// TIA Portal V17 export
// export: Created 2024-08-07T21:44:10.5201385Z, ExportSetting WithDefaults, DisplayName Totally Integrated Automation Portal, DisplayVersion V17 Update 7, DisplayName TIA Portal Openness, DisplayVersion V17 Update 7, DisplayName TIA Portal Version Control Interface, DisplayVersion V17, DisplayName SINAMICS Startdrive Advanced, DisplayVersion V17 SP2, DisplayName SINAMICS Startdrive G110M, G120, G120C, G120D, G120P, G115D, DisplayVersion V17 SP2, DisplayName SINAMICS Startdrive G130, G150, S120, S150, SINAMICS MV, S210, DisplayVersion V17 SP2, DisplayName STEP 7 Professional, DisplayVersion V17 Update 7, DisplayName STEP 7 Safety, DisplayVersion V17 Update 6, DisplayName WinCC Advanced / Unified PC, DisplayVersion V17 Update 7
FUNCTION_BLOCK "1. DMC_setConnection"   // FB2001, LAD
{ S7_Optimized_Access := 'FALSE' }
VERSION : 0.1
// stored: AutoNumber false, IsIECCheckEnabled false, SetENOAutomatically false, UDAEnableTagReadback false
   VAR DB_SPECIFIC
      Connection : Struct
         IPAddress : WString := WSTRING#'';   // IP without the opc.tcp://
         ServerPort : WString := WSTRING#'';   // Only numbers
         PlantID : WString := WSTRING#'';
         PLC_ID : WString := WSTRING#'';
         OperationMode : Bool := False;
      END_STRUCT;
      Controllers : Struct
         opcUaConnect : Bool;
         opcUaMethodCall : Bool;
         opcUaMethodIndex : SInt;
         opcUaConnected { S7_SetPoint := 'True'} : Bool;
         opcUaDone : Bool;
         opcUaBusy : Bool;
         opcUaError : Bool;
         opcUaStatus : Word;
         opcUaDiagnostics : "typeFbDiagnostics";
      END_STRUCT;
      Auxiliar : Struct   // Method fb's call auxiliar variables
         endpointTemp : String[254];
         idx : Int;
         timeout : Bool;
         reconnectionTimeout : Bool;
         tryAgain : Bool;
      END_STRUCT;
      Timers : Struct
         timeoutCallMethod : TON_TIME;
         forceReconnection { S7_SetPoint := 'True'} : TON_TIME;
         tryAgain { S7_SetPoint := 'True'} : TON_TIME;
      END_STRUCT;
      CallBuffer : Array[0..#nMethods] of Bool;
   END_VAR
   VAR_TEMP
      methodInputs : Variant;
      methodOutputs : Variant;
      retVal : Int;
   END_VAR
   VAR CONSTANT
      nMethods : Int := 9;
      callTimeout : Time := T#5s;
   END_VAR
BEGIN

REGION Network 1 (SCL): Set connection
   // Assign data from MII_PARAMETERS [DB2020]
   #Connection.IPAddress := "MII_Parameters".Connection.IPAddress;
   #Connection.ServerPort := "MII_Parameters".Connection.ServerPort;
   #Connection.PlantID := "MII_Parameters".Connection.PlantID;
   #Connection.PLC_ID := "MII_Parameters".Connection.PLC_ID;
   #Connection.OperationMode := "MII_Parameters".Connection.OperationMode;

   // Configure IP + Port to establish connection
   IF "MII_Interface_Configuration".Connection.ServerEndpointUrl <> #Auxiliar.endpointTemp OR #Connection.IPAddress = WSTRING#'' OR #Connection.ServerPort = WSTRING#'' THEN
       #Controllers.opcUaConnect := FALSE;
       #Auxiliar.endpointTemp := "MII_Interface_Configuration".Connection.ServerEndpointUrl;
   ELSE
       "MII_Interface_Configuration".Connection.ServerEndpointUrl := WSTRING_TO_STRING(CONCAT_WSTRING(IN1 := WSTRING#'opc.tcp://', IN2 := #Connection.IPAddress, IN3 := WSTRING#':', IN4 := #Connection.ServerPort, IN5 := WSTRING#'/PCoUaServer'));
       #Controllers.opcUaConnect := TRUE;
   END_IF;

   // Manual reconnection
   IF NOT #Auxiliar.reconnectionTimeout AND "MII_Parameters".Commands.forceReconnection THEN
       #Auxiliar.endpointTemp := String#'';
   END_IF;

   //Force reconnection timer
   #Timers.forceReconnection(IN := "MII_Parameters".Commands.forceReconnection,
   PT := t#2s,
   Q => #Auxiliar.reconnectionTimeout);

   // Reset force reconnection after 2s
   IF #Auxiliar.reconnectionTimeout THEN
       "MII_Parameters".Commands.forceReconnection := FALSE;
   END_IF;

   //Method call timeout
   #Timers.timeoutCallMethod(IN := #Controllers.opcUaMethodCall,
   PT := t#5s,
   Q => #Auxiliar.timeout);
END_REGION

REGION Network 2 (SCL): Prepare method call
   IF #Controllers.opcUaConnected = FALSE THEN
       //DOWNGRADED MODE
       #Controllers.opcUaMethodCall := FALSE;

   ELSE
       //NORMAL MODE
       FOR #Auxiliar.idx := 0 TO #nMethods DO
           IF #Controllers.opcUaMethodCall = FALSE AND #CallBuffer[#Auxiliar.idx] = TRUE THEN
               #Controllers.opcUaMethodIndex := INT_TO_SINT(#Auxiliar.idx);
               #Controllers.opcUaMethodCall := TRUE;
           END_IF;
       END_FOR;

       REGION SWITCH CASE
           CASE #Controllers.opcUaMethodIndex OF
               0:  //M000_PRODUCTION_DECLARATION
                   #methodInputs := REF("MII_Interface_Data".MII_METHODS."M000_PRODUCTION_DECLARATION".Inputs);
                   VariantPut(SRC := "MII_Interface_Data".MII_METHODS."M000_PRODUCTION_DECLARATION".Inputs,
                              DST := #methodInputs);
                   #methodOutputs := REF("MII_Interface_Data".MII_METHODS."M000_PRODUCTION_DECLARATION".Outputs);
                   VariantPut(SRC := "MII_Interface_Data".MII_METHODS."M000_PRODUCTION_DECLARATION".Outputs,
                              DST := #methodOutputs);

               1:  //M001_GET_LOCAL_TIME
                   #methodOutputs := REF("MII_Interface_Data".MII_METHODS."M001_GET_LOCAL_TIME".Outputs);
                   VariantPut(SRC := "MII_Interface_Data".MII_METHODS."M001_GET_LOCAL_TIME".Outputs,
                              DST := #methodOutputs);

               2:  //M101_SCRAP_DECLARATION
                   #methodInputs := REF("MII_Interface_Data".MII_METHODS."M101_SCRAP_DECLARATION".Inputs);
                   VariantPut(SRC := "MII_Interface_Data".MII_METHODS."M101_SCRAP_DECLARATION".Inputs,
                              DST := #methodInputs);
                   #methodOutputs := REF("MII_Interface_Data".MII_METHODS."M101_SCRAP_DECLARATION".Outputs);
                   VariantPut(SRC := "MII_Interface_Data".MII_METHODS."M101_SCRAP_DECLARATION".Outputs,
                              DST := #methodOutputs);

               3:  //M003_GENERATE_ALERT
                   #methodInputs := REF("MII_Interface_Data".MII_METHODS."M003_GENERATE_ALERT".Inputs);
                   VariantPut(SRC := "MII_Interface_Data".MII_METHODS."M003_GENERATE_ALERT".Inputs,
                              DST := #methodInputs);
                   #methodOutputs := REF("MII_Interface_Data".MII_METHODS."M003_GENERATE_ALERT".Outputs);
                   VariantPut(SRC := "MII_Interface_Data".MII_METHODS."M003_GENERATE_ALERT".Outputs,
                              DST := #methodOutputs);

               4:  //M102_REWORK_DECLARATION
                   #methodInputs := REF("MII_Interface_Data".MII_METHODS."M102_REWORK_DECLARATION".Inputs);
                   VariantPut(SRC := "MII_Interface_Data".MII_METHODS."M102_REWORK_DECLARATION".Inputs,
                              DST := #methodInputs);
                   #methodOutputs := REF("MII_Interface_Data".MII_METHODS."M102_REWORK_DECLARATION".Outputs);
                   VariantPut(SRC := "MII_Interface_Data".MII_METHODS."M102_REWORK_DECLARATION".Outputs,
                              DST := #methodOutputs);

               5:  //M002_GET_PLANTS
                   #methodOutputs := REF("MII_Interface_Data".MII_METHODS."M002_GET_PLANTS".Outputs);
                   VariantPut(SRC := "MII_Interface_Data".MII_METHODS.M002_GET_PLANTS.Outputs,
                              DST := #methodOutputs);

               6: //NON TRS
                   #methodInputs := REF("MII_Interface_Data".MII_METHODS.M004_NTRS.Inputs);
                   VariantPut(SRC := "MII_Interface_Data".MII_METHODS.M004_NTRS.Inputs,
                              DST := #methodInputs);
                   #methodOutputs := REF("MII_Interface_Data".MII_METHODS.M004_NTRS.Outputs);
                   VariantPut(SRC := "MII_Interface_Data".MII_METHODS.M004_NTRS.Outputs,
                              DST := #methodOutputs);

               7: //PY
                   #methodInputs := REF("MII_Interface_Data".MII_METHODS.M103_PY.Inputs);
                   VariantPut(SRC := "MII_Interface_Data".MII_METHODS.M103_PY.Inputs,
                              DST := #methodInputs);
                   #methodOutputs := REF("MII_Interface_Data".MII_METHODS.M103_PY.Outputs);
                   VariantPut(SRC := "MII_Interface_Data".MII_METHODS.M103_PY.Outputs,
                              DST := #methodOutputs);

               8: //VARABILITY
                   #methodInputs := REF("MII_Interface_Data".MII_METHODS.M005_VARIABILITY.Inputs);
                   VariantPut(SRC := "MII_Interface_Data".MII_METHODS.M005_VARIABILITY.Inputs,
                              DST := #methodInputs);
                   #methodOutputs := REF("MII_Interface_Data".MII_METHODS.M005_VARIABILITY.Outputs);
                   VariantPut(SRC := "MII_Interface_Data".MII_METHODS.M005_VARIABILITY.Outputs,
                              DST := #methodOutputs);


           END_CASE;
       END_REGION ;
   END_IF;
END_REGION

REGION Network 3: Call client fb
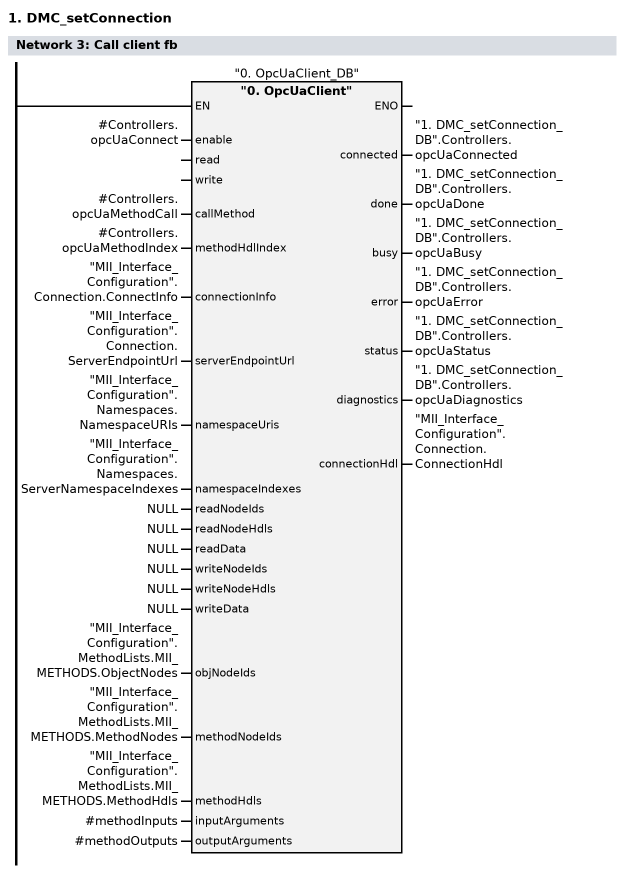
   RUNG wire#powerrail
      "0. OpcUaClient_DB"(enable := #Controllers.opcUaConnect, read :=, write :=, callMethod := #Controllers.opcUaMethodCall, methodHdlIndex := #Controllers.opcUaMethodIndex, connectionInfo := "MII_Interface_Configuration".Connection.ConnectInfo, serverEndpointUrl := "MII_Interface_Configuration".Connection.ServerEndpointUrl, namespaceUris := "MII_Interface_Configuration".Namespaces.NamespaceURIs, namespaceIndexes := "MII_Interface_Configuration".Namespaces.ServerNamespaceIndexes, readNodeIds := NULL, readNodeHdls := NULL, readData := NULL, writeNodeIds := NULL, writeNodeHdls := NULL, writeData := NULL, objNodeIds := "MII_Interface_Configuration".MethodLists.MII_METHODS.ObjectNodes, methodNodeIds := "MII_Interface_Configuration".MethodLists.MII_METHODS.MethodNodes, methodHdls := "MII_Interface_Configuration".MethodLists.MII_METHODS.MethodHdls, inputArguments := #methodInputs, outputArguments := #methodOutputs, connected => "1. DMC_setConnection_DB".Controllers.opcUaConnected, done => "1. DMC_setConnection_DB".Controllers.opcUaDone, busy => "1. DMC_setConnection_DB".Controllers.opcUaBusy, error => "1. DMC_setConnection_DB".Controllers.opcUaError, status => "1. DMC_setConnection_DB".Controllers.opcUaStatus, diagnostics => "1. DMC_setConnection_DB".Controllers.opcUaDiagnostics, connectionHdl => "MII_Interface_Configuration".Connection.ConnectionHdl)
   END_RUNG
   // the same network as SCL:
   "0. OpcUaClient_DB"(enable := #Controllers.opcUaConnect,   // "0. OpcUaClient"
                       callMethod := #Controllers.opcUaMethodCall,
                       methodHdlIndex := #Controllers.opcUaMethodIndex,
                       connectionInfo := "MII_Interface_Configuration".Connection.ConnectInfo,
                       serverEndpointUrl := "MII_Interface_Configuration".Connection.ServerEndpointUrl,
                       namespaceUris := "MII_Interface_Configuration".Namespaces.NamespaceURIs,
                       namespaceIndexes := "MII_Interface_Configuration".Namespaces.ServerNamespaceIndexes,
                       readNodeIds := NULL,
                       readNodeHdls := NULL,
                       readData := NULL,
                       writeNodeIds := NULL,
                       writeNodeHdls := NULL,
                       writeData := NULL,
                       objNodeIds := "MII_Interface_Configuration".MethodLists.MII_METHODS.ObjectNodes,
                       methodNodeIds := "MII_Interface_Configuration".MethodLists.MII_METHODS.MethodNodes,
                       methodHdls := "MII_Interface_Configuration".MethodLists.MII_METHODS.MethodHdls,
                       inputArguments := #methodInputs,
                       outputArguments := #methodOutputs,
                       connected => "1. DMC_setConnection_DB".Controllers.opcUaConnected,
                       done => "1. DMC_setConnection_DB".Controllers.opcUaDone,
                       busy => "1. DMC_setConnection_DB".Controllers.opcUaBusy,
                       error => "1. DMC_setConnection_DB".Controllers.opcUaError,
                       status => "1. DMC_setConnection_DB".Controllers.opcUaStatus,
                       diagnostics => "1. DMC_setConnection_DB".Controllers.opcUaDiagnostics,
                       connectionHdl => "MII_Interface_Configuration".Connection.ConnectionHdl);
END_REGION

REGION Network 4 (SCL): Post method call
   IF #Controllers.opcUaMethodCall AND (#Controllers.opcUaDone OR #Auxiliar.timeout) THEN
       REGION SWITCH CASE
           CASE #Controllers.opcUaMethodIndex OF
               0:  //M000_PRODUCTION_DECLARATION
                   //Send the inputs and the output to the HMI
                   "MII_Parameters".M000_Status.Inputs := "MII_Interface_Data".MII_METHODS.M000_PRODUCTION_DECLARATION.Inputs;
                   "MII_Parameters".M000_Status.Outputs := "MII_Interface_Data".MII_METHODS.M000_PRODUCTION_DECLARATION.Outputs;


                   IF "MII_Interface_Data".MII_METHODS.M000_PRODUCTION_DECLARATION.Outputs.SUCCESS_FLAG = 0 OR #Auxiliar.timeout THEN
                       //Write error status
                       IF #Auxiliar.timeout THEN
                           "MII_Parameters".M000_Status.status := Wstring#'TimeoutERROR';
                       ELSE
                           "MII_Parameters".M000_Status.status := "MII_Interface_Data".MII_METHODS.M000_PRODUCTION_DECLARATION.Outputs.STATUS_MESSAGE;
                       END_IF;

                       //Get error timestamp 
                       #retVal := RD_LOC_T("MII_Parameters".M000_Status.timestamp);

                       //Set error trigger to HMI store values
                       //Note: HMI must reset this tag after writing the file
                       "MII_Parameters".M000_Status.error := TRUE;
                   ELSE
                       //Reset error if declaration is ok
                       "MII_Parameters".M000_Status.error := FALSE;
                       "MII_Parameters".M000_Status.status := "MII_Interface_Data".MII_METHODS.M000_PRODUCTION_DECLARATION.Outputs.STATUS_MESSAGE;
                   END_IF;

                   //Reset test command and add one to the auxiliar cycle counter
                   IF "MII_Parameters".Commands.testProdDeclaration THEN
                       "MII_Parameters".Commands.testProdDeclaration := FALSE;
                       "MII_Parameters".Commands.auxTestProdDeclaration := "MII_Parameters".Commands.auxTestProdDeclaration + 1;
                   END_IF;

               1: //M002_GET_LOCAL_TIME
                   IF #Auxiliar.timeout THEN
                       "MII_Parameters".M002_Status.status := WSTRING#'TimeoutERROR';
                   ELSE
                       //Overwrite system time
                       #retVal := WR_LOC_T(LOCTIME := "MII_Interface_Data".MII_METHODS.M001_GET_LOCAL_TIME.Outputs.DATETIME_LOCAL, DST := TRUE);

                       //Set M002_status
                       "MII_Parameters".M002_Status.localTime := "MII_Interface_Data".MII_METHODS.M001_GET_LOCAL_TIME.Outputs.DATETIME_LOCAL;
                       "MII_Parameters".M002_Status.status := WSTRING#'OK';

                       //Reset command after calling the method
                       "MII_Parameters".Commands.getLocalTime := FALSE;
                   END_IF;

               2: //TO BE DEVELOPED
                   ;

               3: //TO BE DEVELOPED
                   ;

               4: //TO BE DEVELOPED
                   ;

               5: //TO BE DEVELOPED
                   ;

               6: //TO BE DEVELOPED
                   ;

               7: //TO BE DEVELOPED
                   ;

               8: //TO BE DEVELOPED
                   ;

           END_CASE;
       END_REGION

       //RESET METHOD INDEX
       #CallBuffer[#Controllers.opcUaMethodIndex] := FALSE;

       //RESET METHOD TAG
       #Controllers.opcUaMethodCall := FALSE;
   END_IF;
END_REGION

REGION Network 5 (SCL): Device diagnostics
   // Read diagnostic status
   "MII_Parameters".Connection_Status.opcUaConnected := #Controllers.opcUaConnected;
   "MII_Parameters".Connection_Status.opcUaError := #Controllers.opcUaError;
   "MII_Parameters".Connection_Status.opcUaStatus := #Controllers.opcUaStatus;
   "MII_Parameters".Connection_Status.opcUaDiagnostics := #Controllers.opcUaDiagnostics.subfunctionStatus;

   // Shift data to display on HMI
   IF #Controllers.opcUaDiagnostics.subfunctionStatus > 65536 THEN
       "MII_Parameters".Connection_Status.aux.opcUaSubfunctionStatus := SHR(IN := #Controllers.opcUaDiagnostics.subfunctionStatus, N := 16);
   END_IF;

   // Output error parameters
   IF NOT #Controllers.opcUaError THEN
       CASE #Controllers.opcUaStatus OF
           16#0000:
               IF NOT #Controllers.opcUaDone THEN
                   //Client not connected.
                   "MII_Parameters".Connection_Status.aux.diagnosticStatus := 1;
               ELSE
                   //Job successfully executed.
                   "MII_Parameters".Connection_Status.aux.diagnosticStatus := 2;
               END_IF;

           16#7000:
               IF NOT #Controllers.opcUaDone THEN
                   //Client connected and ready for job.
                   "MII_Parameters".Connection_Status.aux.diagnosticStatus := 3;
               ELSE
                   //Connection successfully established and ready for job.
                   "MII_Parameters".Connection_Status.aux.diagnosticStatus := 4;
               END_IF;

           16#7001: //Job is running.
               "MII_Parameters".Connection_Status.aux.diagnosticStatus := 5;
       END_CASE;
   ELSE
       // Output parameters with error
       "MII_Parameters".Connection_Status.aux.diagnosticStatus := #Controllers.opcUaStatus;

       // Automatically manage the 16#80AE_0000 error
       IF NOT "MII_Parameters".Commands.forceReconnection AND NOT "MII_Parameters".Connection_Status.opcUaConnected THEN
           // Forces the reconnection
           "MII_Parameters".Commands.forceReconnection := TRUE;

           IF "0. OpcUaClient_DB".statOpcUaRequests.disconnect THEN
               // Reset disconnect button 
               "0. OpcUaClient_DB".statOpcUaRequests.disconnect := FALSE;
           END_IF;
       END_IF;
   END_IF;
END_REGION

REGION Network 6 (SCL): Try to call method again routine
   // //Method call timeout
   // #Timers.tryAgain(IN := "MII_Parameters".M000_Status.error,
   //                  PT := t#2s,
   //                  Q => #Auxiliar.tryAgain);

   // IF #Controllers.opcUaConnected AND #Auxiliar.tryAgain THEN
   //              //Try again
   //              IF NOT #CallBuffer[0] THEN
   //                  #CallBuffer[0] := TRUE;

   //                  //Add one attempt to counter
   //                  "MII_Parameters".Connection_Status.aux.nAttemptsTotal := "MII_Parameters".Connection_Status.aux.nAttemptsTotal + 1;
   //              END_IF;

   //              //Restart timer
   //              RESET_TIMER(#Timers.tryAgain);

   //          END_IF;
END_REGION
END_FUNCTION_BLOCK
